TEXTLIST AxesDialogSignTextList
  0 = '+'
  1 = '-'
   = ''
END_TEXTLIST

(* stored: Version 1.1.0.1, ProductVersion 3.1.4019.2
   TextList AxesDialogSignTextList: Id {f51266b8-089b-4ea3-a0a4-de7721f66844} *)
